(* PLC project Unnamed, Unknown Unnamed 1 *)
(* stored: creationDateTime 2023-05-11T09:59:03, modificationDateTime 2023-06-07T16:50:25 *)

PROGRAM projek_mekatronika_kompleks
  VAR
    SensorTinggi AT %IX100.0 : BOOL;
    SensorRendah AT %IX100.1 : BOOL;
    SensorPallet AT %IX100.2 : BOOL;
    Loaded AT %IX100.3 : BOOL;
    EntryKiri AT %IX100.4 : BOOL;
    ExitKiri AT %IX100.5 : BOOL;
    EntryKanan AT %IX100.6 : BOOL;
    ExitKanan AT %IX100.7 : BOOL;
    BerhentiDarurat AT %IX100.8 : BOOL;
    Start AT %IX100.9 : BOOL;
    Reset AT %IX100.10 : BOOL;
    Stop AT %IX100.11 : BOOL;
    FactoryBerjalan AT %IX100.12 : BOOL;
    Manual AT %IX100.13 : BOOL;
    Auto AT %IX100.14 : BOOL;
    PalletSensor AT %IX100.15 : BOOL;
    SensorPickPlaceKanan AT %IX100.16 : BOOL;
    SensorRendahKANAN AT %IX100.17 : BOOL;
    SensorTinggiKANAN AT %IX100.18 : BOOL;
    SensorPickPlaceKIRI AT %IX100.19 : BOOL;
    EntryConveyor AT %QX100.0 : BOOL;
    Load AT %QX100.1 : BOOL;
    Unload AT %QX100.2 : BOOL;
    KeKiri AT %QX100.3 : BOOL;
    KeKanan AT %QX100.4 : BOOL;
    ConveyorKiri AT %QX100.5 : BOOL;
    ConveyorKanan AT %QX100.6 : BOOL;
    Emitter AT %QX100.7 : BOOL;
    RemoverKiri AT %QX100.8 : BOOL;
    RemoverKanan AT %QX100.9 : BOOL;
    LampuStart AT %QX100.10 : BOOL;
    LampuReset AT %QX100.11 : BOOL;
    LampuStop AT %QX100.12 : BOOL;
    ConveyorKananBelokKiri AT %QX100.13 : BOOL;
    ConveyorPickPlaceKanan AT %QX100.14 : BOOL;
    AmbilKANAN AT %QX100.15 : BOOL;
    BCKanan AT %QX100.16 : BOOL;
    BCKananNaik AT %QX100.17 : BOOL;
    BCBelokPalletizer AT %QX100.18 : BOOL;
    BCKiri1 AT %QX100.19 : BOOL;
    BCPalletizer AT %QX100.20 : BOOL;
    BCNaikPalletizer AT %QX100.21 : BOOL;
    AmbilKIRI AT %QX100.22 : BOOL;
    AutoMode AT %IX0.0 : BOOL;
    ResetMode AT %IX0.1 : BOOL;
    ManualMode AT %IX0.2 : BOOL;
    RunningMode AT %IX0.3 : BOOL;
    StartLatch AT %IX0.4 : BOOL;
    PalletSensorMem AT %IX0.5 : BOOL;
    SensorRendahMem AT %IX0.6 : BOOL;
    SensorTinggiMem AT %IX0.7 : BOOL;
    SensorRendahReset AT %IX0.8 : BOOL;
    SensorTinggiReset AT %IX0.9 : BOOL;
    SensorRendahKANANMem AT %IX0.10 : BOOL;
    SensorTinggiKANANMem AT %IX0.11 : BOOL;
    PindahBoxKANANMem AT %QX0.0 : BOOL;
    BalikTempatKANANMem AT %QX0.1 : BOOL;
    SensorResetKANAN AT %QX0.2 : BOOL;
    PindahBoxKIRIMem AT %QX0.3 : BOOL;
    BalikTempatKIRIMem AT %QX0.4 : BOOL;
    LepasKiriMem AT %QX0.5 : BOOL;
    PusherReset AT %QX0.6 : BOOL;
    DepanBlkgKANAN AT %QW100 : INT;
    AtasBawahKANAN AT %QW101 : INT;
    KiriKananKANAN AT %QW102 : INT;
    DepanBlkgKIRI AT %QW103 : INT;
    AtasBawahKIRI AT %QW104 : INT;
    KiriKananKIRI AT %QW105 : INT;
    BCKiriNaik1 AT %QW106 : INT;
  END_VAR
  VAR
    TON0 : TON;
    TON1 : TON;
    TON2 : TON;
    TON3 : TON;
    TON4 : TON;
    TON5 : TON;
    TON6 : TON;
    TON7 : TON;
    TON8 : TON;
    TON10 : TON;
    TON11 : TON;
    TON9 : TON;
    TON12 : TON;
    TON13 : TON;
    TON14 : TON;
    TON15 : TON;
    TON16 : TON;
    TON18 : TON;
    TON21 : TON;
    TON24 : TON;
    TON19 : TON;
    TON20 : TON;
    TON22 : TON;
    TON23 : TON;
  END_VAR
  VAR  (* added by the conversion: wires and edge detectors of the diagram *)
    _MOVE271_ENO : BOOL;
    _MOVE271_OUT : INT;
    _MOVE280_ENO : BOOL;
    _MOVE280_OUT : INT;
    _MOVE277_ENO : BOOL;
    _MOVE277_OUT : INT;
    _MOVE317_ENO : BOOL;
    _MOVE317_OUT : INT;
    _MOVE265_ENO : BOOL;
    _MOVE265_OUT : INT;
    _MOVE293_ENO : BOOL;
    _MOVE293_OUT : INT;
    _MOVE305_ENO : BOOL;
    _MOVE305_OUT : INT;
    _MOVE308_ENO : BOOL;
    _MOVE308_OUT : INT;
    _MOVE311_ENO : BOOL;
    _MOVE311_OUT : INT;
    _MOVE121_ENO : BOOL;
    _MOVE121_OUT : INT;
    _MOVE112_ENO : BOOL;
    _MOVE112_OUT : INT;
    _MOVE18_ENO : BOOL;
    _MOVE18_OUT : INT;
    _MOVE195_ENO : BOOL;
    _MOVE195_OUT : INT;
    _MOVE186_ENO : BOOL;
    _MOVE186_OUT : INT;
    _MOVE176_ENO : BOOL;
    _MOVE176_OUT : INT;
    _MOVE81_ENO : BOOL;
    _MOVE81_OUT : INT;
    _MOVE123_ENO : BOOL;
    _MOVE123_OUT : INT;
    _MOVE138_ENO : BOOL;
    _MOVE138_OUT : INT;
    _MOVE181_ENO : BOOL;
    _MOVE181_OUT : INT;
    _MOVE197_ENO : BOOL;
    _MOVE197_OUT : INT;
    _MOVE212_ENO : BOOL;
    _MOVE212_OUT : INT;
    _MOVE142_ENO : BOOL;
    _MOVE142_OUT : INT;
    _MOVE145_ENO : BOOL;
    _MOVE145_OUT : INT;
    _MOVE148_ENO : BOOL;
    _MOVE148_OUT : INT;
    _MOVE216_ENO : BOOL;
    _MOVE216_OUT : INT;
    _MOVE219_ENO : BOOL;
    _MOVE219_OUT : INT;
    _MOVE222_ENO : BOOL;
    _MOVE222_OUT : INT;
  END_VAR

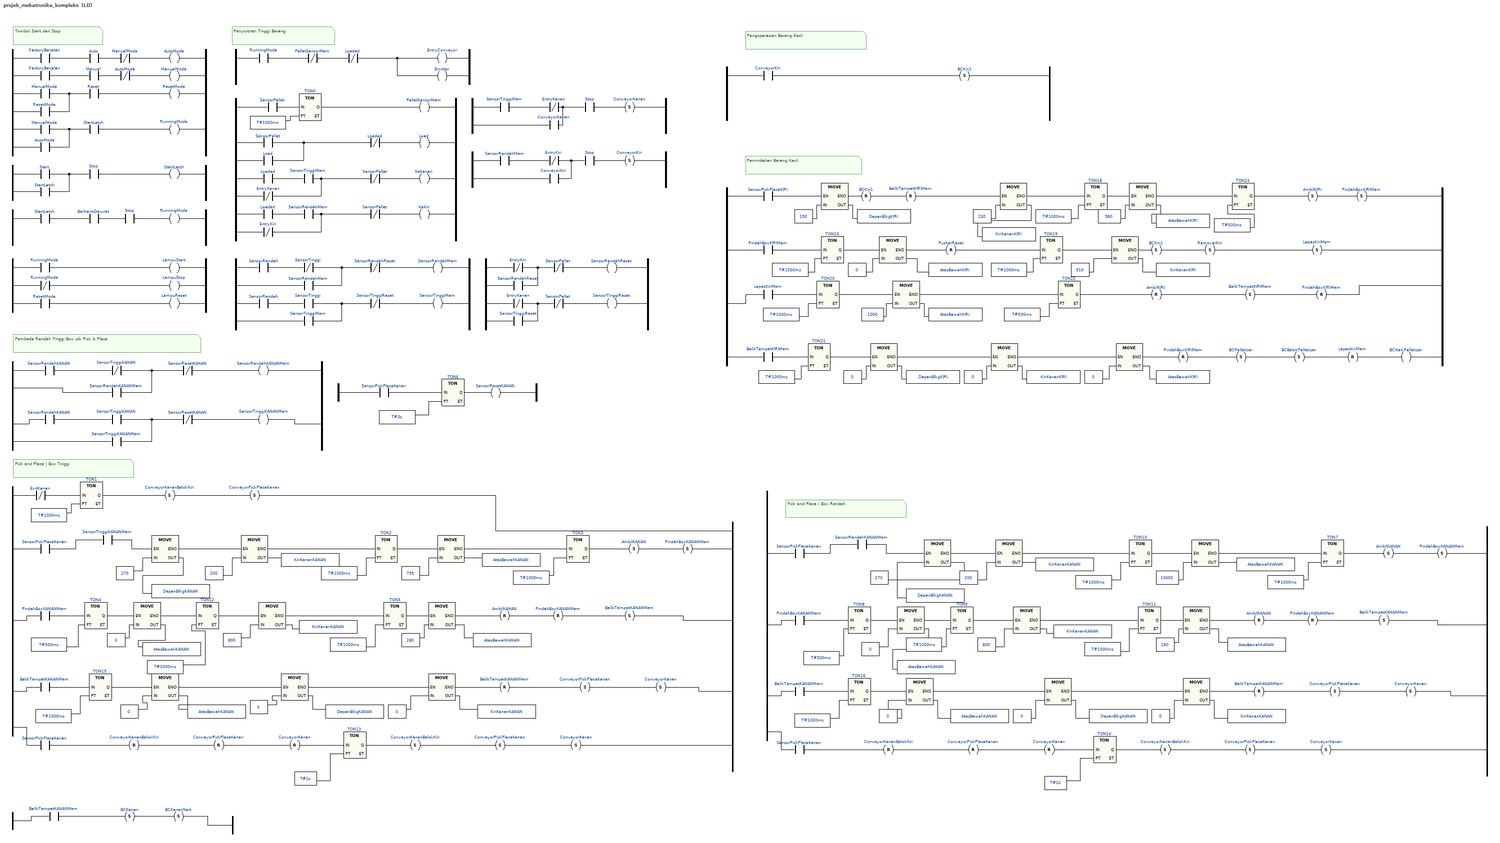
(* LD diagram, written out as Structured Text *)
(* Tombol Start dan Stop *)
(* Penyortiran Tinggi Barang *)
(* Pengoperasian Barang Kecil *)
AutoMode := FactoryBerjalan AND Auto AND NOT ManualMode;
EntryConveyor := RunningMode AND NOT PalletSensorMem AND NOT Loaded;
ManualMode := FactoryBerjalan AND Manual AND NOT AutoMode;
Emitter := RunningMode AND NOT PalletSensorMem AND NOT Loaded;
IF ConveyorKiri THEN BCKiri1 := TRUE; END_IF;
ResetMode := (ManualMode OR ResetMode) AND Reset;
TON0(IN := SensorPallet, PT := T#1000ms);
PalletSensorMem := TON0.Q;
IF (SensorTinggiMem AND NOT EntryKanan OR ConveyorKanan) AND Stop THEN ConveyorKanan := TRUE; END_IF;
RunningMode := (ManualMode OR AutoMode) AND StartLatch;
Load := (Load OR SensorPallet) AND NOT Loaded;
(* Pemindahan Barang Kecil *)
IF (SensorRendahMem AND NOT EntryKiri OR ConveyorKiri) AND Stop THEN ConveyorKiri := TRUE; END_IF;
StartLatch := (StartLatch OR Start) AND Stop;
KeKanan := (NOT EntryKanan OR Loaded AND SensorTinggiMem) AND NOT SensorPallet;
_MOVE271_OUT := MOVE(EN := SensorPickPlaceKIRI, IN := 190, ENO => _MOVE271_ENO);
IF _MOVE271_ENO THEN BCKiri1 := FALSE; END_IF;
IF _MOVE271_ENO THEN BalikTempatKIRIMem := FALSE; END_IF;
_MOVE280_OUT := MOVE(EN := _MOVE271_ENO, IN := 230, ENO => _MOVE280_ENO);
TON18(IN := _MOVE280_ENO, PT := T#1000ms);
_MOVE277_OUT := MOVE(EN := TON18.Q, IN := 980, ENO => _MOVE277_ENO);
TON24(IN := _MOVE277_ENO, PT := T#500ms);
IF TON24.Q THEN AmbilKIRI := TRUE; END_IF;
IF TON24.Q THEN PindahBoxKIRIMem := TRUE; END_IF;
KeKiri := (NOT EntryKiri OR Loaded AND SensorRendahMem) AND NOT SensorPallet;
IF _MOVE271_ENO THEN DepanBlkgKIRI := _MOVE271_OUT; END_IF;
RunningMode := StartLatch AND BerhentiDarurat AND Stop;
IF _MOVE277_ENO THEN AtasBawahKIRI := _MOVE277_OUT; END_IF;
IF _MOVE280_ENO THEN KiriKananKIRI := _MOVE280_OUT; END_IF;
TON23(IN := PindahBoxKIRIMem, PT := T#1000ms);
_MOVE317_OUT := MOVE(EN := TON23.Q, IN := 0, ENO => _MOVE317_ENO);
IF _MOVE317_ENO THEN PusherReset := FALSE; END_IF;
TON19(IN := _MOVE317_ENO, PT := T#1000ms);
_MOVE265_OUT := MOVE(EN := TON19.Q, IN := 910, ENO => _MOVE265_ENO);
IF _MOVE265_ENO THEN BCKiri1 := TRUE; END_IF;
IF _MOVE265_ENO THEN RemoverKiri := TRUE; END_IF;
IF _MOVE265_ENO THEN LepasKiriMem := TRUE; END_IF;
LampuStart := RunningMode;
SensorRendahMem := (SensorRendah AND NOT SensorTinggi OR SensorRendahMem) AND NOT SensorRendahReset;
SensorRendahReset := (SensorRendahReset OR NOT EntryKiri) AND NOT SensorPallet;
IF _MOVE317_ENO THEN AtasBawahKIRI := _MOVE317_OUT; END_IF;
IF _MOVE265_ENO THEN KiriKananKIRI := _MOVE265_OUT; END_IF;
LampuStop := NOT RunningMode;
TON20(IN := LepasKiriMem, PT := T#1000ms);
_MOVE293_OUT := MOVE(EN := TON20.Q, IN := 1000, ENO => _MOVE293_ENO);
TON22(IN := _MOVE293_ENO, PT := T#500ms);
IF TON22.Q THEN AmbilKIRI := FALSE; END_IF;
IF TON22.Q THEN BalikTempatKIRIMem := TRUE; END_IF;
IF TON22.Q THEN PindahBoxKIRIMem := FALSE; END_IF;
LampuReset := ResetMode;
SensorTinggiMem := (SensorTinggiMem OR SensorRendah AND SensorTinggi) AND NOT SensorTinggiReset;
SensorTinggiReset := (NOT EntryKanan OR SensorTinggiReset) AND NOT SensorPallet;
IF _MOVE293_ENO THEN AtasBawahKIRI := _MOVE293_OUT; END_IF;
(* Pembeda Rendah Tinggi Box utk Pick & Place *)
TON21(IN := BalikTempatKIRIMem, PT := T#1000ms);
_MOVE305_OUT := MOVE(EN := TON21.Q, IN := 0, ENO => _MOVE305_ENO);
_MOVE308_OUT := MOVE(EN := _MOVE305_ENO, IN := 0, ENO => _MOVE308_ENO);
_MOVE311_OUT := MOVE(EN := _MOVE308_ENO, IN := 0, ENO => _MOVE311_ENO);
IF _MOVE311_ENO THEN PindahBoxKIRIMem := FALSE; END_IF;
IF _MOVE311_ENO THEN BCPalletizer := TRUE; END_IF;
IF _MOVE311_ENO THEN BCBelokPalletizer := TRUE; END_IF;
IF _MOVE311_ENO THEN LepasKiriMem := FALSE; END_IF;
BCNaikPalletizer := _MOVE311_ENO;
SensorRendahKANANMem := (SensorRendahKANANMem OR SensorRendahKANAN AND NOT SensorTinggiKANAN) AND NOT SensorResetKANAN;
IF _MOVE305_ENO THEN DepanBlkgKIRI := _MOVE305_OUT; END_IF;
IF _MOVE308_ENO THEN KiriKananKIRI := _MOVE308_OUT; END_IF;
IF _MOVE311_ENO THEN AtasBawahKIRI := _MOVE311_OUT; END_IF;
TON6(IN := SensorPickPlaceKanan, PT := T#3s);
SensorResetKANAN := TON6.Q;
SensorTinggiKANANMem := (SensorRendahKANAN AND SensorTinggiKANAN OR SensorTinggiKANANMem) AND NOT SensorResetKANAN;
(* Pick and Place | Box Tinggi *)
TON1(IN := NOT ExitKanan, PT := T#1000ms);
IF TON1.Q THEN ConveyorKananBelokKiri := TRUE; END_IF;
IF TON1.Q THEN ConveyorPickPlaceKanan := TRUE; END_IF;
(* Pick and Place | Box Rendah *)
_MOVE121_OUT := MOVE(EN := SensorPickPlaceKanan AND SensorTinggiKANANMem, IN := 270, ENO => _MOVE121_ENO);
_MOVE112_OUT := MOVE(EN := _MOVE121_ENO, IN := 200, ENO => _MOVE112_ENO);
TON2(IN := _MOVE112_ENO, PT := T#1000ms);
_MOVE18_OUT := MOVE(EN := TON2.Q, IN := 795, ENO => _MOVE18_ENO);
TON3(IN := _MOVE18_ENO, PT := T#1000ms);
IF TON3.Q THEN AmbilKANAN := TRUE; END_IF;
IF TON3.Q THEN PindahBoxKANANMem := TRUE; END_IF;
_MOVE195_OUT := MOVE(EN := SensorPickPlaceKanan AND SensorRendahKANANMem, IN := 270, ENO => _MOVE195_ENO);
_MOVE186_OUT := MOVE(EN := _MOVE195_ENO, IN := 200, ENO => _MOVE186_ENO);
TON10(IN := _MOVE186_ENO, PT := T#1000ms);
_MOVE176_OUT := MOVE(EN := TON10.Q, IN := 10000, ENO => _MOVE176_ENO);
TON7(IN := _MOVE176_ENO, PT := T#1000ms);
IF TON7.Q THEN AmbilKANAN := TRUE; END_IF;
IF TON7.Q THEN PindahBoxKANANMem := TRUE; END_IF;
IF _MOVE112_ENO THEN KiriKananKANAN := _MOVE112_OUT; END_IF;
IF _MOVE18_ENO THEN AtasBawahKANAN := _MOVE18_OUT; END_IF;
IF _MOVE186_ENO THEN KiriKananKANAN := _MOVE186_OUT; END_IF;
IF _MOVE176_ENO THEN AtasBawahKANAN := _MOVE176_OUT; END_IF;
IF _MOVE121_ENO THEN DepanBlkgKANAN := _MOVE121_OUT; END_IF;
IF _MOVE195_ENO THEN DepanBlkgKANAN := _MOVE195_OUT; END_IF;
TON4(IN := PindahBoxKANANMem, PT := T#500ms);
_MOVE81_OUT := MOVE(EN := TON4.Q, IN := 0, ENO => _MOVE81_ENO);
TON12(IN := _MOVE81_ENO, PT := T#2000ms);
_MOVE123_OUT := MOVE(EN := TON12.Q, IN := 800, ENO => _MOVE123_ENO);
TON5(IN := _MOVE123_ENO, PT := T#1000ms);
_MOVE138_OUT := MOVE(EN := TON5.Q, IN := 280, ENO => _MOVE138_ENO);
IF _MOVE138_ENO THEN AmbilKANAN := FALSE; END_IF;
IF _MOVE138_ENO THEN PindahBoxKANANMem := FALSE; END_IF;
IF _MOVE138_ENO THEN BalikTempatKANANMem := TRUE; END_IF;
TON8(IN := PindahBoxKANANMem, PT := T#500ms);
_MOVE181_OUT := MOVE(EN := TON8.Q, IN := 0, ENO => _MOVE181_ENO);
TON9(IN := _MOVE181_ENO, PT := T#1000ms);
_MOVE197_OUT := MOVE(EN := TON9.Q, IN := 800, ENO => _MOVE197_ENO);
TON11(IN := _MOVE197_ENO, PT := T#1000ms);
_MOVE212_OUT := MOVE(EN := TON11.Q, IN := 280, ENO => _MOVE212_ENO);
IF _MOVE212_ENO THEN AmbilKANAN := FALSE; END_IF;
IF _MOVE212_ENO THEN PindahBoxKANANMem := FALSE; END_IF;
IF _MOVE212_ENO THEN BalikTempatKANANMem := TRUE; END_IF;
IF _MOVE123_ENO THEN KiriKananKANAN := _MOVE123_OUT; END_IF;
IF _MOVE197_ENO THEN KiriKananKANAN := _MOVE197_OUT; END_IF;
IF _MOVE138_ENO THEN AtasBawahKANAN := _MOVE138_OUT; END_IF;
IF _MOVE212_ENO THEN AtasBawahKANAN := _MOVE212_OUT; END_IF;
IF _MOVE81_ENO THEN AtasBawahKANAN := _MOVE81_OUT; END_IF;
IF _MOVE181_ENO THEN AtasBawahKANAN := _MOVE181_OUT; END_IF;
TON15(IN := BalikTempatKANANMem, PT := T#1000ms);
_MOVE142_OUT := MOVE(EN := TON15.Q, IN := 0, ENO => _MOVE142_ENO);
_MOVE145_OUT := MOVE(EN := _MOVE142_ENO, IN := 0, ENO => _MOVE145_ENO);
_MOVE148_OUT := MOVE(EN := _MOVE145_ENO, IN := 0, ENO => _MOVE148_ENO);
IF _MOVE148_ENO THEN BalikTempatKANANMem := FALSE; END_IF;
IF _MOVE148_ENO THEN ConveyorPickPlaceKanan := TRUE; END_IF;
IF _MOVE148_ENO THEN ConveyorKanan := TRUE; END_IF;
TON16(IN := BalikTempatKANANMem, PT := T#1000ms);
_MOVE216_OUT := MOVE(EN := TON16.Q, IN := 0, ENO => _MOVE216_ENO);
_MOVE219_OUT := MOVE(EN := _MOVE216_ENO, IN := 0, ENO => _MOVE219_ENO);
_MOVE222_OUT := MOVE(EN := _MOVE219_ENO, IN := 0, ENO => _MOVE222_ENO);
IF _MOVE222_ENO THEN BalikTempatKANANMem := FALSE; END_IF;
IF _MOVE222_ENO THEN ConveyorPickPlaceKanan := TRUE; END_IF;
IF _MOVE222_ENO THEN ConveyorKanan := TRUE; END_IF;
IF _MOVE142_ENO THEN AtasBawahKANAN := _MOVE142_OUT; END_IF;
IF _MOVE145_ENO THEN DepanBlkgKANAN := _MOVE145_OUT; END_IF;
IF _MOVE148_ENO THEN KiriKananKANAN := _MOVE148_OUT; END_IF;
IF _MOVE216_ENO THEN AtasBawahKANAN := _MOVE216_OUT; END_IF;
IF _MOVE219_ENO THEN DepanBlkgKANAN := _MOVE219_OUT; END_IF;
IF _MOVE222_ENO THEN KiriKananKANAN := _MOVE222_OUT; END_IF;
IF SensorPickPlaceKanan THEN ConveyorKananBelokKiri := FALSE; END_IF;
IF SensorPickPlaceKanan THEN ConveyorPickPlaceKanan := FALSE; END_IF;
IF SensorPickPlaceKanan THEN ConveyorKanan := FALSE; END_IF;
TON13(IN := SensorPickPlaceKanan, PT := T#2s);
IF TON13.Q THEN ConveyorKananBelokKiri := TRUE; END_IF;
IF TON13.Q THEN ConveyorPickPlaceKanan := TRUE; END_IF;
IF TON13.Q THEN ConveyorKanan := TRUE; END_IF;
IF SensorPickPlaceKanan THEN ConveyorKananBelokKiri := FALSE; END_IF;
IF SensorPickPlaceKanan THEN ConveyorPickPlaceKanan := FALSE; END_IF;
IF SensorPickPlaceKanan THEN ConveyorKanan := FALSE; END_IF;
TON14(IN := SensorPickPlaceKanan, PT := T#2s);
IF TON14.Q THEN ConveyorKananBelokKiri := TRUE; END_IF;
IF TON14.Q THEN ConveyorPickPlaceKanan := TRUE; END_IF;
IF TON14.Q THEN ConveyorKanan := TRUE; END_IF;
IF BalikTempatKANANMem THEN BCKanan := TRUE; END_IF;
IF BalikTempatKANANMem THEN BCKananNaik := TRUE; END_IF;
END_PROGRAM

CONFIGURATION Config0
  RESOURCE Res0 ON PLC
    TASK task0(INTERVAL := T#20ms, PRIORITY := 0);
    PROGRAM instance0 WITH task0 : projek_mekatronika_kompleks;
  END_RESOURCE
END_CONFIGURATION
